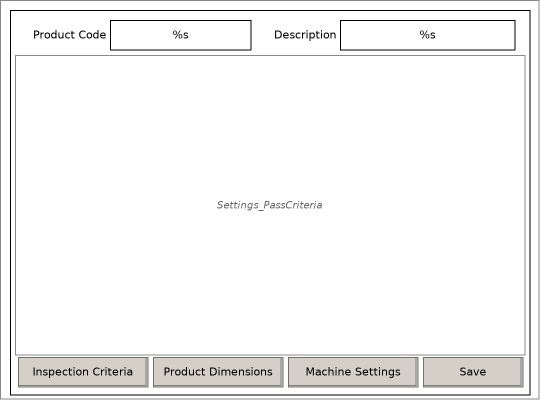
VISUALIZATION SettingsTemplate  // 540x400
VAR_IN_OUT
	Tube : ST_TubeParameters;
END_VAR
    Rectangle (10,10 520x385)
    Rectangle (110,20 141x30), "%s", text variable: Tube.ProductName
        OnMouseClick: write Tube.ProductName via Default
    Label (30,20 80x30), "Product Code"
    Button (288,357 130x30), "Machine Settings"
        OnMouseClick: FrameSelectionChange Selection=SelectedFrame=c09837a4-7cd0-42f3-a923-2461df8b3e92, Selection=1, GlobSel=AssignType=Directly, SelType=Locally
    Button (18,357 130x30), "Inspection Criteria"
        OnMouseClick: FrameSelectionChange Selection=SelectedFrame=c09837a4-7cd0-42f3-a923-2461df8b3e92, GlobSel=AssignType=Directly, SelType=Locally
    Button (153,357 130x30), "Product Dimensions"
        OnMouseClick: FrameSelectionChange Selection=SelectedFrame=c09837a4-7cd0-42f3-a923-2461df8b3e92, Selection=2, GlobSel=AssignType=Directly, SelType=Locally
    Button (423,357 100x30), "Save"
        OnMouseClick: execute { MAIN.bSave := TRUE; }
    Frame (15,55 510x300)
        shows Settings_PassCriteria(CutHeightMin := Tube.MinHeight, CutHeightMax := Tube.MaxHeight, CutLengthMin := Tube.MinLength, CutLengthMax := Tube.MaxLength, CutToleranceX := Tube.ResultToleranceX, CutToleranceY := Tube.ResultToleranceY, AdjustmentX := Tube.AdjustmentX, AdjustmentY := Tube.AdjustmentY, AdjustmentLength := Tube.AdjustmentLength)
        shows Settings_Mandrel(CutPositionX := Tube.CutPositionX, CutPositionY := Tube.CutPositionY, InspectPositionX := Tube.InspectPositionX, InspectPositionY := Tube.InspectPositionY, EjectPositionX := Tube.EjectPositionX, EjectPositionY := Tube.EjectPositionY, VacuumThreshold := Tube.VacuumThreshold, VacuumPosition := Tube.VacPosition)
        shows Settings_ProductDimensions(Diameter := Tube.Diameter, PocketDepth := Tube.DepthOfPocket)
    Label (271,20 69x30), "Description"
    Rectangle (340,20 175x30), "%s", text variable: Tube.Description
        OnMouseClick: write Tube.Description via Default
END_VISUALIZATION

(* stored: Version 1.1.0.1, ProductVersion 3.1.4024.9
   Visu SettingsTemplate: Id {faa4d7a8-9daa-42ca-89dd-62d087bb12b6} *)
